# EPICS autosave request: softGlueApp/Db/FreqCntr_settings.req
$(P)$(H)FreqCntr-$(N)_desc
$(P)$(H)FreqCntr-$(N)_CLK_Signal
